Staubli VAL3: loadNextOne.pgx

program loadNextOne(string x_sName)
begin
  prog_swap:libLoad(x_sName)
end
